FUNCTION_BLOCK SocketRecieveTask IMPLEMENTS ITask
VAR_INPUT
END_VAR
VAR_OUTPUT
	rxBuffer : ARRAY[0..1439] OF BYTE;
END_VAR
VAR
	iState: INT;
	_done: BOOL;
	_busy: BOOL;
	_error: BOOL;
	_execute: BOOL;
	fbSocketRecieve : Tc2_TcpIp.FB_SocketReceive;
	
	fbReceiveTimer : Tc2_Standard.TON;
END_VAR

CASE iState OF
	0:
		IF _execute THEN
			_done := FALSE;
			_busy := TRUE;
			_error := FALSE;
			iState := 5;
			_execute := FALSE;
		END_IF
		
	5:	
		fbReceiveTimer.IN := TRUE;
		fbSocketRecieve.bExecute := TRUE;
		IF fbReceiveTimer.Q THEN
			iState := 10;
			fbReceiveTimer.IN := FALSE;
		END_IF
	10:
		fbSocketRecieve.bExecute := FALSE;
		IF NOT fbSocketRecieve.bBusy THEN
			IF NOT fbSocketRecieve.bError THEN
				IF (fbSocketRecieve.nRecBytes > 0) THEN
					_busy := FALSE;
					_done := TRUE;
					iState := 0;
				ELSE
					iState := 5;
				END_IF
			ELSE
				_error := TRUE;
				_busy := FALSE;
				fbSocketRecieve.bExecute := FALSE;
				iState := 0;
			END_IF
			
		END_IF
END_CASE
fbReceiveTimer(PT := T#100MS);
fbSocketRecieve(pDest := ADR(rxBuffer),
				cbLen := SIZEOF(rxBuffer),
				tTimeout := Tc2_System.DEFAULT_ADS_TIMEOUT);

METHOD Abort : BOOL
fbSocketRecieve.bExecute := FALSE;
_busy := FALSE;
_execute := FALSE;
Abort := TRUE;
iState := 0;
END_METHOD

PROPERTY Busy : BOOL
GET
Busy := _busy;
END_GET
END_PROPERTY

PROPERTY Done : BOOL
GET
Done := _done;
END_GET
END_PROPERTY

PROPERTY Error : BOOL
GET
Error := _error;
END_GET
END_PROPERTY

METHOD Execute : BOOL
IF NOT fbSocketRecieve.bBusy THEN
	Execute := _execute := true;
END_IF
END_METHOD

PROPERTY PUBLIC RemoteSocket : T_HSOCKET
GET // PUBLIC
RemoteSocket := fbSocketRecieve.hSocket;
END_GET
SET // PUBLIC
fbSocketRecieve.hSocket := RemoteSocket;
END_SET
END_PROPERTY

END_FUNCTION_BLOCK

(* stored: Version 1.1.0.1, ProductVersion 3.1.4024.12
   POU SocketRecieveTask: Id {e15ca270-1c0a-48bd-83a0-101e82ff50ce}, SpecialFunc None
   Method Abort: Id {c73408db-da2b-404e-8fa3-3d61894ae1a3}
   Property Busy: Id {dba5f978-5ec6-4ff4-9c27-f3474ca48bc3}
   Get Get: Id {c1260c39-6a85-4ccc-a013-642999cf6c71}
   Property Done: Id {b2a0b8c3-3507-4e85-9295-1f62288504d6}
   Get Get: Id {e1f2c216-7440-4bac-b40b-0240942d2cd5}
   Property Error: Id {2a95e621-93aa-4241-8d57-8085e6017400}
   Get Get: Id {23764fb3-8e61-43c0-a8c5-6d1c5a4cff34}
   Method Execute: Id {0552173e-02fe-4343-8acd-3a31e9bcf1e5}
   Property RemoteSocket: Id {20bfcffa-39ed-4ef5-88bc-7beef535c9f6}
   Get Get: Id {51a9adc8-0e16-4e31-b92b-2feac3dcef53}
   Set Set: Id {f5d4dfeb-b5ea-49a8-bd39-f798943c2dbe} *)
